// TIA Portal V17 export
// export: Created 2024-09-02T12:50:33.2303231Z, ExportSetting WithDefaults, DisplayName Totally Integrated Automation Portal, DisplayVersion V17, DisplayName TIA Portal Openness, DisplayVersion V17, DisplayName TIA Portal Version Control Interface, DisplayVersion V17, DisplayName STEP 7 Professional, DisplayVersion V17, DisplayName STEP 7 Safety, DisplayVersion V17, DisplayName WinCC Professional, DisplayVersion V17
TYPE "Omron_PLC_Test"
// stored: IsFailsafeCompliant false
   STRUCT
      "Controle_Output(2Words)" : Struct
         Chanel0 : Struct
            Flg : Bool;
            Busy : Bool;
            Reserve_0_2 : Bool;
            "OR" : Bool;
            Run : Bool;
            Reserve_0_5 : Bool;
            Reserve_0_6 : Bool;
            Reserve_0_7 : Bool;
            XFlag : Bool;
            Xbusy : Bool;
            xWait : Bool;
            Reserve_1_3 : Bool;
            Reserve_1_4 : Bool;
            Reserve_1_5 : Bool;
            Reserve_1_6 : Bool;
            Err : Bool;
         END_STRUCT;
         Chanel1 : Struct
            Gate : Bool;
            Reserve_2_1 : Bool;
            Reserve_2_2 : Bool;
            Reserve_2_3 : Bool;
            Reserve_2_4 : Bool;
            Reserve_2_5 : Bool;
            Reserve_2_6 : Bool;
            Reserve_2_7 : Bool;
            Reserve_3_0 : Bool;
            Reserve_3_1 : Bool;
            Reserve_3_2 : Bool;
            Reserve_3_3 : Bool;
            Reserve_3_4 : Bool;
            Reserve_3_5 : Bool;
            Reserve_3_6 : Bool;
            Reserve_3_7 : Bool;
         END_STRUCT;
      END_STRUCT;
   END_STRUCT;
END_TYPE
